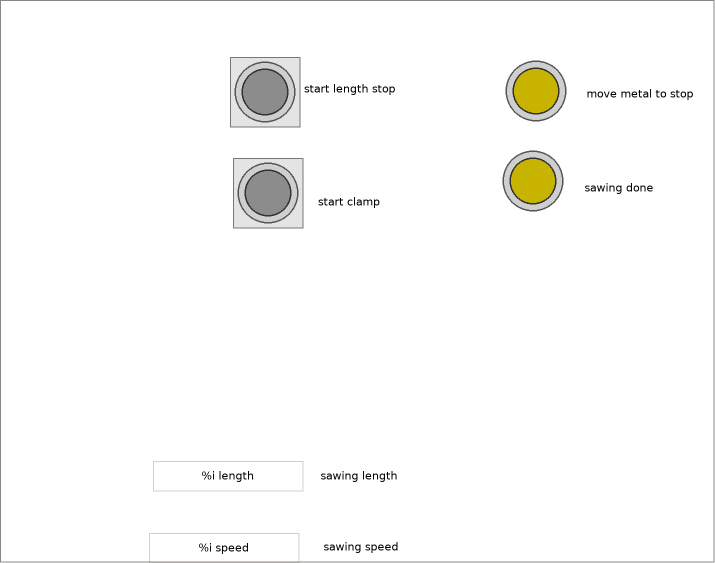
VISUALIZATION Visualization_1  // 715x563
    PushSwitch (230,57 70x70), variable: POU_UserInterface.startButtonLengthStop, behaviour: TOGGLE, style: Switch-PushSwitch-Gray
    PushSwitch (233,158 70x70), variable: POU_UserInterface.startClamp, behaviour: TOGGLE, style: Switch-PushSwitch-Gray
    Lamp1 (501,56 70x70), variable: POU_UserInterface.messageMoveMetalToStop, style: Lamp-Lamp1-Yellow
    Lamp1 (498,146 70x70), variable: POU_UserInterface.sawingDone, style: Lamp-Lamp1-Yellow
    Textfield (153,461 150x30), "%i length", text variable: POU_UserInterface.sawingLength
        OnMouseClick: write the text variable via Default
    Textfield (149,533 150x30), "%i speed", text variable: POU_UserInterface.sawingSpeed
        OnMouseClick: write the text variable via Default
    Label (565,79 150x30), "move metal to stop"
    Label (544,173 150x30), "sawing done"
    Label (274,187 150x30), "start clamp"
    Label (284,461 150x30), "sawing length"
    Label (275,74 150x30), "start length stop"
    Label (286,532 150x30), "sawing speed"
END_VISUALIZATION

(* stored: Version 1.1.0.1, ProductVersion 3.1.4024.12
   Visu Visualization_1: Id {b767637b-73f3-43cc-8e82-5650a0d8700a} *)
